// TIA Portal V20 export
DATA_BLOCK "HmiInterface"   // DB159
// stored: Access Published, MemoryReserve 100, Namespace Unit1.Em3
   VAR
      em : "LAF_typeEmInterface";
      cm : "Unit1.Em3.typeCmHmiInterface";
      topTapeLoading : "LER_typeSequenceInterface";
      topTapeAttachment : "LER_typeSequenceInterface";
      topTapeFixStage : "LER_typeSequenceInterface";
      TopTapeIdleTime : "Unit1.Em3.typeTopTapeIdleTimeHmiInterface";
      topTapeCuttingCount : "LER_typeAlarmCounterInterface";
      cmTopTapeJRDetect : "LBC_typeDigitalSignalInterface";
      cmTopTapeDiameter : "LBC_typeDigitalSignalInterface";
   END_VAR
   VAR RETAIN
      cmTopTapeAxisX { S7_SetPoint := 'True'} : "LBC_typeAxis64PosInterface";
      cmTopTapeAxisY { S7_SetPoint := 'True'} : "LBC_typeAxis64PosInterface";
   END_VAR
   VAR
      cmTopTapeLoadingBwdFwd : "LBC_typeTwoWayActuatorInterface";
      cmTopTapeLoadingClampOpenClose : "LBC_typeTwoWayActuatorInterface";
      cmTopTapeCutterUpDown : "LBC_typeTwoWayActuatorInterface";
      cmTopTapeCutterClampUpDown : "LBC_typeTwoWayActuatorInterface";
      cmTopTapeTensionBwdFwd : "LBC_typeTwoWayActuatorInterface";
      cmTopTapeAttachmentUpDown : "LBC_typeTwoWayActuatorInterface";
      cmTopTapeClampTopLeftUpDown : "LBC_typeTwoWayActuatorInterface";
      cmTopTapeClampTopCenterUpDown : "LBC_typeTwoWayActuatorInterface";
      cmTopTapeClampTopRightUpDown : "LBC_typeTwoWayActuatorInterface";
      cmTopTapeClampBtmDownUp : "LBC_typeTwoWayActuatorInterface";
      cmTopTapeClampAllOpenClose : "LBC_typeTwoWayActuatorInterface";
      cmTopTapeAttachmentVaccumOffOn : "LBC_typeTwoWayActuatorInterface";
      cmQrHandyReader : "LER_typeDM8700Interface";
      intCondition : "Unit1.Em3.typeIntConditionHmiInterface";
   END_VAR
BEGIN
   em.interlinkMode.link := FALSE;
   em.interlinkMode.unlink := FALSE;
   em.interlinkMode.isLinked := TRUE;
   em.commands.enable := FALSE;
   em.commands.acknowledge := FALSE;
   em.commands.disableAlarms := FALSE;
   em.commands.activateSimulation := FALSE;
   em.commands.home := FALSE;
   em.commands.moveToInitialPosition := FALSE;
   em.commands.directModeControl := 16#0000_0002;
   em.commands.directStateControl := 16#0000_0002;
   em.status.enabled := FALSE;
   em.status.acknowledgeActive := FALSE;
   em.status.alarmsDisabled := FALSE;
   em.status.simulationActive := FALSE;
   em.status.safetyReleased := TRUE;
   em.status.initialized := FALSE;
   em.status.homed := TRUE;
   em.status.safeState := FALSE;
   em.status.stateComplete := FALSE;
   em.alarms.error := FALSE;
   em.alarms.warning := FALSE;
   em.alarms.info := FALSE;
   TopTapeIdleTime.processCount := T#300M;
   topTapeCuttingCount.referenceDesignator := WSTRING#'Em3 Top Tape Cutting Count';
   topTapeCuttingCount.ProcessValue.faultCount := 50000;
   topTapeCuttingCount.SetValue.faultCount := 50000;
   cmTopTapeJRDetect.commands.refreshConfiguration := FALSE;
   cmTopTapeJRDetect.commands.editConfiguration := FALSE;
   cmTopTapeJRDetect.commands.saveConfiguration := FALSE;
   cmTopTapeJRDetect.commands.reset := FALSE;
   cmTopTapeJRDetect.monitoring.enable := TRUE;
   cmTopTapeJRDetect.monitoring.referenceDesignator := WSTRING#'DigitalSignal';
   cmTopTapeJRDetect.monitoring.simulation := FALSE;
   cmTopTapeJRDetect.monitoring.processValue := FALSE;
   cmTopTapeJRDetect.monitoring.error := FALSE;
   cmTopTapeJRDetect.monitoring.status := 16#0000;
   cmTopTapeJRDetect.configuration.referenceDesignator := WSTRING#'DigitalSignal';
   cmTopTapeJRDetect.configuration.onDelay := T#0MS;
   cmTopTapeJRDetect.configuration.offDelay := T#0MS;
   cmTopTapeJRDetect.configuration.default := FALSE;
   cmTopTapeJRDetect.configuration.invertProcessValue := FALSE;
   cmTopTapeJRDetect.configuration.disableAlarms := FALSE;
   cmTopTapeDiameter.commands.refreshConfiguration := FALSE;
   cmTopTapeDiameter.commands.editConfiguration := FALSE;
   cmTopTapeDiameter.commands.saveConfiguration := FALSE;
   cmTopTapeDiameter.commands.reset := FALSE;
   cmTopTapeDiameter.monitoring.enable := TRUE;
   cmTopTapeDiameter.monitoring.referenceDesignator := WSTRING#'DigitalSignal';
   cmTopTapeDiameter.monitoring.simulation := FALSE;
   cmTopTapeDiameter.monitoring.processValue := FALSE;
   cmTopTapeDiameter.monitoring.error := FALSE;
   cmTopTapeDiameter.monitoring.status := 16#0000;
   cmTopTapeDiameter.configuration.referenceDesignator := WSTRING#'DigitalSignal';
   cmTopTapeDiameter.configuration.onDelay := T#0MS;
   cmTopTapeDiameter.configuration.offDelay := T#0MS;
   cmTopTapeDiameter.configuration.default := FALSE;
   cmTopTapeDiameter.configuration.invertProcessValue := FALSE;
   cmTopTapeDiameter.configuration.disableAlarms := FALSE;
   cmTopTapeAxisX.commandConfiguration.generalSettings.stopOnError := TRUE;
   cmTopTapeAxisX.commandConfiguration.generalSettings.resetWithRestart := FALSE;
   cmTopTapeAxisX.commandConfiguration.generalSettings.abortWaitingSyncCmd := TRUE;
   cmTopTapeAxisX.commandConfiguration.power.startMode := 1;
   cmTopTapeAxisX.commandConfiguration.power.stopMode := 0;
   cmTopTapeAxisX.commandConfiguration.power.syncMotionSimulation := FALSE;
   cmTopTapeAxisX.commandConfiguration.power.syncMotionSimulationExtendedMode := -1;
   cmTopTapeAxisX.commandConfiguration.jog.velocity := 1.0;
   cmTopTapeAxisX.commandConfiguration.jog.acceleration := 100.0;
   cmTopTapeAxisX.commandConfiguration.jog.deceleration := 100.0;
   cmTopTapeAxisX.commandConfiguration.jog.jerk := 0.0;
   cmTopTapeAxisX.commandConfiguration.jog.positionControlled := TRUE;
   cmTopTapeAxisX.commandConfiguration.jog.increment := 0.0;
   cmTopTapeAxisX.commandConfiguration.jog.mode := 0;
   cmTopTapeAxisX.commandConfiguration.moveVelocity.velocity := 10.0;
   cmTopTapeAxisX.commandConfiguration.moveVelocity.acceleration := 1000.0;
   cmTopTapeAxisX.commandConfiguration.moveVelocity.deceleration := 1000.0;
   cmTopTapeAxisX.commandConfiguration.moveVelocity.jerk := -1.0;
   cmTopTapeAxisX.commandConfiguration.moveVelocity.direction := 0;
   cmTopTapeAxisX.commandConfiguration.moveVelocity.positionControlled := TRUE;
   cmTopTapeAxisX.commandConfiguration.moveVelocity.velocityChangeOnTheFly := FALSE;
   cmTopTapeAxisX.commandConfiguration.stop.deceleration := -1.0;
   cmTopTapeAxisX.commandConfiguration.stop.jerk := -1.0;
   cmTopTapeAxisX.commandConfiguration.stop.abortAcceleration := FALSE;
   cmTopTapeAxisX.commandConfiguration.fastStop.deceleration := -1.0;
   cmTopTapeAxisX.commandConfiguration.fastStop.jerk := -1.0;
   cmTopTapeAxisX.commandConfiguration.fastStop.abortAcceleration := FALSE;
   cmTopTapeAxisX.commandConfiguration.fastStop.replaceStopPossible := FALSE;
   cmTopTapeAxisX.commandConfiguration.torqueLimiting.limit := -1.0;
   cmTopTapeAxisX.commandConfiguration.torqueLimiting.mode := 0;
   cmTopTapeAxisX.commandConfiguration.homing.position := 0.0;
   cmTopTapeAxisX.commandConfiguration.homing.mode := 3;
   cmTopTapeAxisX.commandConfiguration.homing.sensor := 0;
   cmTopTapeAxisX.commandConfiguration.homing.extendedMode := -1;
   cmTopTapeAxisX.commandConfiguration.homing.extendedModeTorqueLimit := 0.0;
   cmTopTapeAxisX.commandConfiguration.homing.extendedModeTargetPosition := 0.0;
   cmTopTapeAxisX.commandConfiguration.posRelative.distance := 0.0;
   cmTopTapeAxisX.commandConfiguration.posRelative.velocity := -1.0;
   cmTopTapeAxisX.commandConfiguration.posRelative.acceleration := -1.0;
   cmTopTapeAxisX.commandConfiguration.posRelative.deceleration := -1.0;
   cmTopTapeAxisX.commandConfiguration.posRelative.jerk := -1.0;
   cmTopTapeAxisX.commandConfiguration.posRelative.direction := 0;
   cmTopTapeAxisX.commandConfiguration.posAbsolute.position := 0.0;
   cmTopTapeAxisX.commandConfiguration.posAbsolute.velocity := -1.0;
   cmTopTapeAxisX.commandConfiguration.posAbsolute.acceleration := -1.0;
   cmTopTapeAxisX.commandConfiguration.posAbsolute.deceleration := -1.0;
   cmTopTapeAxisX.commandConfiguration.posAbsolute.jerk := -1.0;
   cmTopTapeAxisX.commandConfiguration.posAbsolute.direction := 1;
   cmTopTapeAxisX.commandConfiguration.posAbsolute.positionChangeOnTheFly := FALSE;
   cmTopTapeAxisX.commandConfiguration.posAbsolute.velocityChangeOnTheFly := FALSE;
   cmTopTapeAxisX.commandConfiguration.posSuperimposed.distance := 0.0;
   cmTopTapeAxisX.commandConfiguration.posSuperimposed.velocityDiff := -1.0;
   cmTopTapeAxisX.commandConfiguration.posSuperimposed.acceleration := -1.0;
   cmTopTapeAxisX.commandConfiguration.posSuperimposed.deceleration := -1.0;
   cmTopTapeAxisX.commandConfiguration.posSuperimposed.jerk := -1.0;
   cmTopTapeAxisX.commandConfiguration.posSuperimposed.direction := 0;
   cmTopTapeAxisX.commandConfiguration.haltSuperimposed.deceleration := -1.0;
   cmTopTapeAxisX.commandConfiguration.haltSuperimposed.jerk := -1.0;
   cmTopTapeAxisX.commandConfiguration.haltSuperimposed.abortAcceleration := FALSE;
   cmTopTapeAxisX.commandConfiguration.gearInRelative.ratioNumerator := 1;
   cmTopTapeAxisX.commandConfiguration.gearInRelative.ratioDenominator := 1;
   cmTopTapeAxisX.commandConfiguration.gearInRelative.acceleration := -1.0;
   cmTopTapeAxisX.commandConfiguration.gearInRelative.deceleration := -1.0;
   cmTopTapeAxisX.commandConfiguration.gearInRelative.jerk := -1.0;
   cmTopTapeAxisX.commandConfiguration.gearInRelative.ratioChangeOnTheFly := FALSE;
   cmTopTapeAxisX.commandConfiguration.gearInAbsolute.ratioNumerator := 1;
   cmTopTapeAxisX.commandConfiguration.gearInAbsolute.ratioDenominator := 1;
   cmTopTapeAxisX.commandConfiguration.gearInAbsolute.masterSyncPosition := 0.0;
   cmTopTapeAxisX.commandConfiguration.gearInAbsolute.slaveSyncPosition := 0.0;
   cmTopTapeAxisX.commandConfiguration.gearInAbsolute.syncProfileReference := 1;
   cmTopTapeAxisX.commandConfiguration.gearInAbsolute.masterStartDistance := 0.0;
   cmTopTapeAxisX.commandConfiguration.gearInAbsolute.velocity := -1.0;
   cmTopTapeAxisX.commandConfiguration.gearInAbsolute.acceleration := -1.0;
   cmTopTapeAxisX.commandConfiguration.gearInAbsolute.deceleration := -1.0;
   cmTopTapeAxisX.commandConfiguration.gearInAbsolute.jerk := -1.0;
   cmTopTapeAxisX.commandConfiguration.gearInAbsolute.syncDirection := 1;
   cmTopTapeAxisX.commandConfiguration.gearInAbsolute.ratioChangeOnTheFly := FALSE;
   cmTopTapeAxisX.commandConfiguration.gearInVelocity.continuousUpdate := FALSE;
   cmTopTapeAxisX.commandConfiguration.gearInVelocity.ratioNumerator := 1;
   cmTopTapeAxisX.commandConfiguration.gearInVelocity.ratioDenominator := 1;
   cmTopTapeAxisX.commandConfiguration.gearInVelocity.acceleration := -1.0;
   cmTopTapeAxisX.commandConfiguration.gearInVelocity.deceleration := -1.0;
   cmTopTapeAxisX.commandConfiguration.gearInVelocity.jerk := -1.0;
   cmTopTapeAxisX.commandConfiguration.gearInVelocity.positionControlled := FALSE;
   cmTopTapeAxisX.commandConfiguration.camIn.masterOffset := 0.0;
   cmTopTapeAxisX.commandConfiguration.camIn.slaveOffset := 0.0;
   cmTopTapeAxisX.commandConfiguration.camIn.masterScaling := 1.0;
   cmTopTapeAxisX.commandConfiguration.camIn.slaveScaling := 1.0;
   cmTopTapeAxisX.commandConfiguration.camIn.masterSyncPosition := 0.0;
   cmTopTapeAxisX.commandConfiguration.camIn.syncProfileReference := 1;
   cmTopTapeAxisX.commandConfiguration.camIn.masterStartDistance := 0.0;
   cmTopTapeAxisX.commandConfiguration.camIn.velocity := -1.0;
   cmTopTapeAxisX.commandConfiguration.camIn.acceleration := -1.0;
   cmTopTapeAxisX.commandConfiguration.camIn.deceleration := -1.0;
   cmTopTapeAxisX.commandConfiguration.camIn.jerk := -1.0;
   cmTopTapeAxisX.commandConfiguration.camIn.applicationMode := 0;
   cmTopTapeAxisX.commandConfiguration.camIn.syncDirection := 1;
   cmTopTapeAxisX.commandConfiguration.gearOutCamOut.slavePosition := 0.0;
   cmTopTapeAxisX.commandConfiguration.gearOutCamOut.syncProfileReference := 1;
   cmTopTapeAxisX.commandConfiguration.gearOutCamOut.masterStopDistance := 0.0;
   cmTopTapeAxisX.commandConfiguration.gearOutCamOut.deceleration := -1.0;
   cmTopTapeAxisX.commandConfiguration.gearOutCamOut.jerk := -1.0;
   cmTopTapeAxisX.commandConfiguration.gearOutCamOut.syncOutDirection := 3;
   cmTopTapeAxisX.commandConfiguration.gearOutCamOut.gearOutCamOutMode := -1;
   cmTopTapeAxisX.commandConfiguration.phasing.phaseShift := 0.0;
   cmTopTapeAxisX.commandConfiguration.phasing.velocity := -1.0;
   cmTopTapeAxisX.commandConfiguration.phasing.acceleration := -1.0;
   cmTopTapeAxisX.commandConfiguration.phasing.deceleration := -1.0;
   cmTopTapeAxisX.commandConfiguration.phasing.jerk := -1.0;
   cmTopTapeAxisX.commandConfiguration.phasing.profileReference := 0;
   cmTopTapeAxisX.commandConfiguration.phasing.phasingDistance := 0.0;
   cmTopTapeAxisX.commandConfiguration.phasing.startPosition := 0.0;
   cmTopTapeAxisX.commandConfiguration.phasing.direction := 3;
   cmTopTapeAxisX.commandConfiguration.phasing.phaseAbsolute := TRUE;
   cmTopTapeAxisX.commandConfiguration.phasing.phaseShiftChangeOnTheFly := FALSE;
   cmTopTapeAxisX.commandConfiguration.offset.offset := 0.0;
   cmTopTapeAxisX.commandConfiguration.offset.profileReference := 1;
   cmTopTapeAxisX.commandConfiguration.offset.offsetDistance := 0.0;
   cmTopTapeAxisX.commandConfiguration.offset.startPosition := 0.0;
   cmTopTapeAxisX.commandConfiguration.offset.direction := 3;
   cmTopTapeAxisX.commandConfiguration.offset.offsetAbsolute := TRUE;
   cmTopTapeAxisX.commandConfiguration.offset.offsetChangeOnTheFly := FALSE;
   cmTopTapeAxisX.commands.enableMasterControl := FALSE;
   cmTopTapeAxisX.commands.enableAxis := FALSE;
   cmTopTapeAxisX.commands.resetAxis := FALSE;
   cmTopTapeAxisX.commands.openBrake := FALSE;
   cmTopTapeAxisX.commands.jogForward := FALSE;
   cmTopTapeAxisX.commands.jogBackward := FALSE;
   cmTopTapeAxisX.commands.moveVelocity := FALSE;
   cmTopTapeAxisX.commands.stop := FALSE;
   cmTopTapeAxisX.commands.fastStop := FALSE;
   cmTopTapeAxisX.commands.torqueLimiting := FALSE;
   cmTopTapeAxisX.commands.homing := FALSE;
   cmTopTapeAxisX.commands.posRelative := FALSE;
   cmTopTapeAxisX.commands.posAbsolute := FALSE;
   cmTopTapeAxisX.commands.posSuperimposed := FALSE;
   cmTopTapeAxisX.commands.haltSuperimposed := FALSE;
   cmTopTapeAxisX.commands.selectSetPosition := 0;
   cmTopTapeAxisX.commands.uploadParameters := FALSE;
   cmTopTapeAxisX.commands.refreshConfiguration := FALSE;
   cmTopTapeAxisX.commands.editConfiguration := FALSE;
   cmTopTapeAxisX.commands.saveConfiguration := FALSE;
   cmTopTapeAxisX.commands.uploadCurrentTorque := FALSE;
   cmTopTapeAxisX.commands.reset := FALSE;
   cmTopTapeAxisX.monitoring.enable := TRUE;
   cmTopTapeAxisX.monitoring.referenceDesignator := WSTRING#'TOP TAPING X-Axis';
   cmTopTapeAxisX.monitoring.enabled := TRUE;
   cmTopTapeAxisX.monitoring.enableManualCmds := TRUE;
   cmTopTapeAxisX.monitoring.reset := FALSE;
   cmTopTapeAxisX.monitoring.resetAxis := FALSE;
   cmTopTapeAxisX.monitoring.enableAxis := FALSE;
   cmTopTapeAxisX.monitoring.openBrake := FALSE;
   cmTopTapeAxisX.monitoring.jogBackward := FALSE;
   cmTopTapeAxisX.monitoring.jogForward := FALSE;
   cmTopTapeAxisX.monitoring.moveVelocity := FALSE;
   cmTopTapeAxisX.monitoring.stop := FALSE;
   cmTopTapeAxisX.monitoring.fastStop := FALSE;
   cmTopTapeAxisX.monitoring.torqueLimiting := FALSE;
   cmTopTapeAxisX.monitoring.homing := FALSE;
   cmTopTapeAxisX.monitoring.posRelative := FALSE;
   cmTopTapeAxisX.monitoring.posAbsolute := TRUE;
   cmTopTapeAxisX.monitoring.posSuperimposed := FALSE;
   cmTopTapeAxisX.monitoring.haltSuperimposed := FALSE;
   cmTopTapeAxisX.monitoring.brakeOpened := FALSE;
   cmTopTapeAxisX.monitoring.axisEnabled := FALSE;
   cmTopTapeAxisX.monitoring.resetActive := FALSE;
   cmTopTapeAxisX.monitoring.inVelocity := FALSE;
   cmTopTapeAxisX.monitoring.inLimitation := FALSE;
   cmTopTapeAxisX.monitoring.inClamping := FALSE;
   cmTopTapeAxisX.monitoring.startSync := FALSE;
   cmTopTapeAxisX.monitoring.inSync := FALSE;
   cmTopTapeAxisX.monitoring.inSimulation := FALSE;
   cmTopTapeAxisX.monitoring.jogSelected := FALSE;
   cmTopTapeAxisX.monitoring.moveVelocitySelected := FALSE;
   cmTopTapeAxisX.monitoring.stopSelected := FALSE;
   cmTopTapeAxisX.monitoring.fastStopSelected := FALSE;
   cmTopTapeAxisX.monitoring.torqueLimitingSelected := FALSE;
   cmTopTapeAxisX.monitoring.homingSelected := FALSE;
   cmTopTapeAxisX.monitoring.posRelativeSelected := FALSE;
   cmTopTapeAxisX.monitoring.posAbsoluteSelected := TRUE;
   cmTopTapeAxisX.monitoring.posSuperimposedSelected := FALSE;
   cmTopTapeAxisX.monitoring.haltSuperimposedSelected := FALSE;
   cmTopTapeAxisX.monitoring.commandBusy := FALSE;
   cmTopTapeAxisX.monitoring.commandDone := TRUE;
   cmTopTapeAxisX.monitoring.commandAborted := FALSE;
   cmTopTapeAxisX.monitoring.homingCommandBusy := FALSE;
   cmTopTapeAxisX.monitoring.homingCommandDone := FALSE;
   cmTopTapeAxisX.monitoring.homingCommandAborted := FALSE;
   cmTopTapeAxisX.monitoring.superimposedBusy := FALSE;
   cmTopTapeAxisX.monitoring.superimposedDone := FALSE;
   cmTopTapeAxisX.monitoring.superimposedAborted := FALSE;
   cmTopTapeAxisX.monitoring.selectSetPosition := 0;
   cmTopTapeAxisX.monitoring.selectionController := FALSE;
   cmTopTapeAxisX.monitoring.interlockGeneral := FALSE;
   cmTopTapeAxisX.monitoring.interlockJogForward := TRUE;
   cmTopTapeAxisX.monitoring.interlockJogBackward := TRUE;
   cmTopTapeAxisX.monitoring.interlockWarningGeneral := FALSE;
   cmTopTapeAxisX.monitoring.interlockWarningJogForward := FALSE;
   cmTopTapeAxisX.monitoring.interlockWarningJogBackward := FALSE;
   cmTopTapeAxisX.monitoring.valid := TRUE;
   cmTopTapeAxisX.monitoring.busy := TRUE;
   cmTopTapeAxisX.monitoring.error := FALSE;
   cmTopTapeAxisX.monitoring.status := 16#7101;
   cmTopTapeAxisX.monitoring.subfunctionStatus := 16#0000;
   cmTopTapeAxisX.monitoring.actualPosition := -0.999;
   cmTopTapeAxisX.monitoring.actualSpeed := 0.0;
   cmTopTapeAxisX.monitoring.speedUnit := 1062;
   cmTopTapeAxisX.monitoring.positionUnit := 1013;
   cmTopTapeAxisX.monitoring.axisType := 1;
   cmTopTapeAxisX.monitoring.maxVelocity := 1000.0;
   cmTopTapeAxisX.monitoring.actualCurrent := 0.0;
   cmTopTapeAxisX.monitoring.actualTorque := 0.0;
   cmTopTapeAxisX.monitoring.velocityOverrideEnabled := FALSE;
   cmTopTapeAxisX.monitoring.sinaParaError := FALSE;
   cmTopTapeAxisX.monitoring.sinaParaStatus := 16#0000_0000;
   cmTopTapeAxisX.configuration.referenceDesignator := WSTRING#'TOP TAPING X-Axis';
   cmTopTapeAxisX.configuration.disableAlarms := FALSE;
   cmTopTapeAxisX.configuration.masterControlPopUp := TRUE;
   cmTopTapeAxisX.configuration.setPositions[3..9].position := 0.0;
   cmTopTapeAxisX.configuration.setPositions[11..15].position := 0.0;
   cmTopTapeAxisX.configuration.setPositions[3..9].velocity := 0.0;
   cmTopTapeAxisX.configuration.setPositions[11..15].velocity := 0.0;
   cmTopTapeAxisX.configuration.setPositions[3..9].acceleration := 0.0;
   cmTopTapeAxisX.configuration.setPositions[11..15].acceleration := 0.0;
   cmTopTapeAxisX.configuration.setPositions[3..9].deceleration := 0.0;
   cmTopTapeAxisX.configuration.setPositions[11..15].deceleration := 0.0;
   cmTopTapeAxisX.configuration.setPositions[0]."name" := 'Wait [Tape Get]';
   cmTopTapeAxisX.configuration.setPositions[1]."name" := 'Tape1 Put';
   cmTopTapeAxisX.configuration.setPositions[2]."name" := 'Tape2 Put';
   cmTopTapeAxisX.configuration.setPositions[3]."name" := 'Remain Attachment';
   cmTopTapeAxisX.configuration.setPositions[4..8]."name" := '';
   cmTopTapeAxisX.configuration.setPositions[9]."name" := 'tapePutZone';
   cmTopTapeAxisX.configuration.setPositions[10]."name" := 'Tape Put Zone';
   cmTopTapeAxisX.configuration.setPositions[11..15]."name" := '';
   cmTopTapeAxisY.commandConfiguration.generalSettings.stopOnError := TRUE;
   cmTopTapeAxisY.commandConfiguration.generalSettings.resetWithRestart := FALSE;
   cmTopTapeAxisY.commandConfiguration.generalSettings.abortWaitingSyncCmd := TRUE;
   cmTopTapeAxisY.commandConfiguration.power.startMode := 1;
   cmTopTapeAxisY.commandConfiguration.power.stopMode := 0;
   cmTopTapeAxisY.commandConfiguration.power.syncMotionSimulation := FALSE;
   cmTopTapeAxisY.commandConfiguration.power.syncMotionSimulationExtendedMode := -1;
   cmTopTapeAxisY.commandConfiguration.jog.velocity := 20.0;
   cmTopTapeAxisY.commandConfiguration.jog.acceleration := 200.0;
   cmTopTapeAxisY.commandConfiguration.jog.deceleration := 200.0;
   cmTopTapeAxisY.commandConfiguration.jog.jerk := 0.0;
   cmTopTapeAxisY.commandConfiguration.jog.positionControlled := TRUE;
   cmTopTapeAxisY.commandConfiguration.jog.increment := 0.0;
   cmTopTapeAxisY.commandConfiguration.jog.mode := 0;
   cmTopTapeAxisY.commandConfiguration.moveVelocity.velocity := 1.0;
   cmTopTapeAxisY.commandConfiguration.moveVelocity.acceleration := -1.0;
   cmTopTapeAxisY.commandConfiguration.moveVelocity.deceleration := -1.0;
   cmTopTapeAxisY.commandConfiguration.moveVelocity.jerk := -1.0;
   cmTopTapeAxisY.commandConfiguration.moveVelocity.direction := 0;
   cmTopTapeAxisY.commandConfiguration.moveVelocity.positionControlled := TRUE;
   cmTopTapeAxisY.commandConfiguration.moveVelocity.velocityChangeOnTheFly := FALSE;
   cmTopTapeAxisY.commandConfiguration.stop.deceleration := -1.0;
   cmTopTapeAxisY.commandConfiguration.stop.jerk := -1.0;
   cmTopTapeAxisY.commandConfiguration.stop.abortAcceleration := FALSE;
   cmTopTapeAxisY.commandConfiguration.fastStop.deceleration := -1.0;
   cmTopTapeAxisY.commandConfiguration.fastStop.jerk := -1.0;
   cmTopTapeAxisY.commandConfiguration.fastStop.abortAcceleration := FALSE;
   cmTopTapeAxisY.commandConfiguration.fastStop.replaceStopPossible := FALSE;
   cmTopTapeAxisY.commandConfiguration.torqueLimiting.limit := -1.0;
   cmTopTapeAxisY.commandConfiguration.torqueLimiting.mode := 0;
   cmTopTapeAxisY.commandConfiguration.homing.position := 0.0;
   cmTopTapeAxisY.commandConfiguration.homing.mode := 3;
   cmTopTapeAxisY.commandConfiguration.homing.sensor := 0;
   cmTopTapeAxisY.commandConfiguration.homing.extendedMode := -1;
   cmTopTapeAxisY.commandConfiguration.homing.extendedModeTorqueLimit := 0.0;
   cmTopTapeAxisY.commandConfiguration.homing.extendedModeTargetPosition := 0.0;
   cmTopTapeAxisY.commandConfiguration.posRelative.distance := 0.0;
   cmTopTapeAxisY.commandConfiguration.posRelative.velocity := -1.0;
   cmTopTapeAxisY.commandConfiguration.posRelative.acceleration := -1.0;
   cmTopTapeAxisY.commandConfiguration.posRelative.deceleration := -1.0;
   cmTopTapeAxisY.commandConfiguration.posRelative.jerk := -1.0;
   cmTopTapeAxisY.commandConfiguration.posRelative.direction := 0;
   cmTopTapeAxisY.commandConfiguration.posAbsolute.position := 0.0;
   cmTopTapeAxisY.commandConfiguration.posAbsolute.velocity := -1.0;
   cmTopTapeAxisY.commandConfiguration.posAbsolute.acceleration := -1.0;
   cmTopTapeAxisY.commandConfiguration.posAbsolute.deceleration := -1.0;
   cmTopTapeAxisY.commandConfiguration.posAbsolute.jerk := -1.0;
   cmTopTapeAxisY.commandConfiguration.posAbsolute.direction := 1;
   cmTopTapeAxisY.commandConfiguration.posAbsolute.positionChangeOnTheFly := FALSE;
   cmTopTapeAxisY.commandConfiguration.posAbsolute.velocityChangeOnTheFly := FALSE;
   cmTopTapeAxisY.commandConfiguration.posSuperimposed.distance := 0.0;
   cmTopTapeAxisY.commandConfiguration.posSuperimposed.velocityDiff := -1.0;
   cmTopTapeAxisY.commandConfiguration.posSuperimposed.acceleration := -1.0;
   cmTopTapeAxisY.commandConfiguration.posSuperimposed.deceleration := -1.0;
   cmTopTapeAxisY.commandConfiguration.posSuperimposed.jerk := -1.0;
   cmTopTapeAxisY.commandConfiguration.posSuperimposed.direction := 0;
   cmTopTapeAxisY.commandConfiguration.haltSuperimposed.deceleration := -1.0;
   cmTopTapeAxisY.commandConfiguration.haltSuperimposed.jerk := -1.0;
   cmTopTapeAxisY.commandConfiguration.haltSuperimposed.abortAcceleration := FALSE;
   cmTopTapeAxisY.commandConfiguration.gearInRelative.ratioNumerator := 1;
   cmTopTapeAxisY.commandConfiguration.gearInRelative.ratioDenominator := 1;
   cmTopTapeAxisY.commandConfiguration.gearInRelative.acceleration := -1.0;
   cmTopTapeAxisY.commandConfiguration.gearInRelative.deceleration := -1.0;
   cmTopTapeAxisY.commandConfiguration.gearInRelative.jerk := -1.0;
   cmTopTapeAxisY.commandConfiguration.gearInRelative.ratioChangeOnTheFly := FALSE;
   cmTopTapeAxisY.commandConfiguration.gearInAbsolute.ratioNumerator := 1;
   cmTopTapeAxisY.commandConfiguration.gearInAbsolute.ratioDenominator := 1;
   cmTopTapeAxisY.commandConfiguration.gearInAbsolute.masterSyncPosition := 0.0;
   cmTopTapeAxisY.commandConfiguration.gearInAbsolute.slaveSyncPosition := 0.0;
   cmTopTapeAxisY.commandConfiguration.gearInAbsolute.syncProfileReference := 1;
   cmTopTapeAxisY.commandConfiguration.gearInAbsolute.masterStartDistance := 0.0;
   cmTopTapeAxisY.commandConfiguration.gearInAbsolute.velocity := -1.0;
   cmTopTapeAxisY.commandConfiguration.gearInAbsolute.acceleration := -1.0;
   cmTopTapeAxisY.commandConfiguration.gearInAbsolute.deceleration := -1.0;
   cmTopTapeAxisY.commandConfiguration.gearInAbsolute.jerk := -1.0;
   cmTopTapeAxisY.commandConfiguration.gearInAbsolute.syncDirection := 1;
   cmTopTapeAxisY.commandConfiguration.gearInAbsolute.ratioChangeOnTheFly := FALSE;
   cmTopTapeAxisY.commandConfiguration.gearInVelocity.continuousUpdate := FALSE;
   cmTopTapeAxisY.commandConfiguration.gearInVelocity.ratioNumerator := 1;
   cmTopTapeAxisY.commandConfiguration.gearInVelocity.ratioDenominator := 1;
   cmTopTapeAxisY.commandConfiguration.gearInVelocity.acceleration := -1.0;
   cmTopTapeAxisY.commandConfiguration.gearInVelocity.deceleration := -1.0;
   cmTopTapeAxisY.commandConfiguration.gearInVelocity.jerk := -1.0;
   cmTopTapeAxisY.commandConfiguration.gearInVelocity.positionControlled := FALSE;
   cmTopTapeAxisY.commandConfiguration.camIn.masterOffset := 0.0;
   cmTopTapeAxisY.commandConfiguration.camIn.slaveOffset := 0.0;
   cmTopTapeAxisY.commandConfiguration.camIn.masterScaling := 1.0;
   cmTopTapeAxisY.commandConfiguration.camIn.slaveScaling := 1.0;
   cmTopTapeAxisY.commandConfiguration.camIn.masterSyncPosition := 0.0;
   cmTopTapeAxisY.commandConfiguration.camIn.syncProfileReference := 1;
   cmTopTapeAxisY.commandConfiguration.camIn.masterStartDistance := 0.0;
   cmTopTapeAxisY.commandConfiguration.camIn.velocity := -1.0;
   cmTopTapeAxisY.commandConfiguration.camIn.acceleration := -1.0;
   cmTopTapeAxisY.commandConfiguration.camIn.deceleration := -1.0;
   cmTopTapeAxisY.commandConfiguration.camIn.jerk := -1.0;
   cmTopTapeAxisY.commandConfiguration.camIn.applicationMode := 0;
   cmTopTapeAxisY.commandConfiguration.camIn.syncDirection := 1;
   cmTopTapeAxisY.commandConfiguration.gearOutCamOut.slavePosition := 0.0;
   cmTopTapeAxisY.commandConfiguration.gearOutCamOut.syncProfileReference := 1;
   cmTopTapeAxisY.commandConfiguration.gearOutCamOut.masterStopDistance := 0.0;
   cmTopTapeAxisY.commandConfiguration.gearOutCamOut.deceleration := -1.0;
   cmTopTapeAxisY.commandConfiguration.gearOutCamOut.jerk := -1.0;
   cmTopTapeAxisY.commandConfiguration.gearOutCamOut.syncOutDirection := 3;
   cmTopTapeAxisY.commandConfiguration.gearOutCamOut.gearOutCamOutMode := -1;
   cmTopTapeAxisY.commandConfiguration.phasing.phaseShift := 0.0;
   cmTopTapeAxisY.commandConfiguration.phasing.velocity := -1.0;
   cmTopTapeAxisY.commandConfiguration.phasing.acceleration := -1.0;
   cmTopTapeAxisY.commandConfiguration.phasing.deceleration := -1.0;
   cmTopTapeAxisY.commandConfiguration.phasing.jerk := -1.0;
   cmTopTapeAxisY.commandConfiguration.phasing.profileReference := 0;
   cmTopTapeAxisY.commandConfiguration.phasing.phasingDistance := 0.0;
   cmTopTapeAxisY.commandConfiguration.phasing.startPosition := 0.0;
   cmTopTapeAxisY.commandConfiguration.phasing.direction := 3;
   cmTopTapeAxisY.commandConfiguration.phasing.phaseAbsolute := TRUE;
   cmTopTapeAxisY.commandConfiguration.phasing.phaseShiftChangeOnTheFly := FALSE;
   cmTopTapeAxisY.commandConfiguration.offset.offset := 0.0;
   cmTopTapeAxisY.commandConfiguration.offset.profileReference := 1;
   cmTopTapeAxisY.commandConfiguration.offset.offsetDistance := 0.0;
   cmTopTapeAxisY.commandConfiguration.offset.startPosition := 0.0;
   cmTopTapeAxisY.commandConfiguration.offset.direction := 3;
   cmTopTapeAxisY.commandConfiguration.offset.offsetAbsolute := TRUE;
   cmTopTapeAxisY.commandConfiguration.offset.offsetChangeOnTheFly := FALSE;
   cmTopTapeAxisY.commands.enableMasterControl := FALSE;
   cmTopTapeAxisY.commands.enableAxis := FALSE;
   cmTopTapeAxisY.commands.resetAxis := FALSE;
   cmTopTapeAxisY.commands.openBrake := FALSE;
   cmTopTapeAxisY.commands.jogForward := FALSE;
   cmTopTapeAxisY.commands.jogBackward := FALSE;
   cmTopTapeAxisY.commands.moveVelocity := FALSE;
   cmTopTapeAxisY.commands.stop := FALSE;
   cmTopTapeAxisY.commands.fastStop := FALSE;
   cmTopTapeAxisY.commands.torqueLimiting := FALSE;
   cmTopTapeAxisY.commands.homing := FALSE;
   cmTopTapeAxisY.commands.posRelative := FALSE;
   cmTopTapeAxisY.commands.posAbsolute := FALSE;
   cmTopTapeAxisY.commands.posSuperimposed := FALSE;
   cmTopTapeAxisY.commands.haltSuperimposed := FALSE;
   cmTopTapeAxisY.commands.selectSetPosition := 0;
   cmTopTapeAxisY.commands.uploadParameters := FALSE;
   cmTopTapeAxisY.commands.refreshConfiguration := FALSE;
   cmTopTapeAxisY.commands.editConfiguration := FALSE;
   cmTopTapeAxisY.commands.saveConfiguration := FALSE;
   cmTopTapeAxisY.commands.uploadCurrentTorque := FALSE;
   cmTopTapeAxisY.commands.reset := FALSE;
   cmTopTapeAxisY.monitoring.enable := TRUE;
   cmTopTapeAxisY.monitoring.referenceDesignator := WSTRING#'TOP TAPING Y-Axis';
   cmTopTapeAxisY.monitoring.enabled := TRUE;
   cmTopTapeAxisY.monitoring.enableManualCmds := TRUE;
   cmTopTapeAxisY.monitoring.reset := FALSE;
   cmTopTapeAxisY.monitoring.resetAxis := FALSE;
   cmTopTapeAxisY.monitoring.enableAxis := FALSE;
   cmTopTapeAxisY.monitoring.openBrake := FALSE;
   cmTopTapeAxisY.monitoring.jogBackward := FALSE;
   cmTopTapeAxisY.monitoring.jogForward := FALSE;
   cmTopTapeAxisY.monitoring.moveVelocity := FALSE;
   cmTopTapeAxisY.monitoring.stop := FALSE;
   cmTopTapeAxisY.monitoring.fastStop := FALSE;
   cmTopTapeAxisY.monitoring.torqueLimiting := FALSE;
   cmTopTapeAxisY.monitoring.homing := FALSE;
   cmTopTapeAxisY.monitoring.posRelative := FALSE;
   cmTopTapeAxisY.monitoring.posAbsolute := TRUE;
   cmTopTapeAxisY.monitoring.posSuperimposed := FALSE;
   cmTopTapeAxisY.monitoring.haltSuperimposed := FALSE;
   cmTopTapeAxisY.monitoring.brakeOpened := FALSE;
   cmTopTapeAxisY.monitoring.axisEnabled := FALSE;
   cmTopTapeAxisY.monitoring.resetActive := FALSE;
   cmTopTapeAxisY.monitoring.inVelocity := FALSE;
   cmTopTapeAxisY.monitoring.inLimitation := FALSE;
   cmTopTapeAxisY.monitoring.inClamping := FALSE;
   cmTopTapeAxisY.monitoring.startSync := FALSE;
   cmTopTapeAxisY.monitoring.inSync := FALSE;
   cmTopTapeAxisY.monitoring.inSimulation := FALSE;
   cmTopTapeAxisY.monitoring.jogSelected := FALSE;
   cmTopTapeAxisY.monitoring.moveVelocitySelected := FALSE;
   cmTopTapeAxisY.monitoring.stopSelected := FALSE;
   cmTopTapeAxisY.monitoring.fastStopSelected := FALSE;
   cmTopTapeAxisY.monitoring.torqueLimitingSelected := FALSE;
   cmTopTapeAxisY.monitoring.homingSelected := FALSE;
   cmTopTapeAxisY.monitoring.posRelativeSelected := FALSE;
   cmTopTapeAxisY.monitoring.posAbsoluteSelected := TRUE;
   cmTopTapeAxisY.monitoring.posSuperimposedSelected := FALSE;
   cmTopTapeAxisY.monitoring.haltSuperimposedSelected := FALSE;
   cmTopTapeAxisY.monitoring.commandBusy := FALSE;
   cmTopTapeAxisY.monitoring.commandDone := TRUE;
   cmTopTapeAxisY.monitoring.commandAborted := FALSE;
   cmTopTapeAxisY.monitoring.homingCommandBusy := FALSE;
   cmTopTapeAxisY.monitoring.homingCommandDone := FALSE;
   cmTopTapeAxisY.monitoring.homingCommandAborted := FALSE;
   cmTopTapeAxisY.monitoring.superimposedBusy := FALSE;
   cmTopTapeAxisY.monitoring.superimposedDone := FALSE;
   cmTopTapeAxisY.monitoring.superimposedAborted := FALSE;
   cmTopTapeAxisY.monitoring.selectSetPosition := 0;
   cmTopTapeAxisY.monitoring.selectionController := FALSE;
   cmTopTapeAxisY.monitoring.interlockGeneral := FALSE;
   cmTopTapeAxisY.monitoring.interlockJogForward := TRUE;
   cmTopTapeAxisY.monitoring.interlockJogBackward := TRUE;
   cmTopTapeAxisY.monitoring.interlockWarningGeneral := FALSE;
   cmTopTapeAxisY.monitoring.interlockWarningJogForward := FALSE;
   cmTopTapeAxisY.monitoring.interlockWarningJogBackward := FALSE;
   cmTopTapeAxisY.monitoring.valid := TRUE;
   cmTopTapeAxisY.monitoring.busy := TRUE;
   cmTopTapeAxisY.monitoring.error := FALSE;
   cmTopTapeAxisY.monitoring.status := 16#7101;
   cmTopTapeAxisY.monitoring.subfunctionStatus := 16#0000;
   cmTopTapeAxisY.monitoring.actualPosition := 293.001;
   cmTopTapeAxisY.monitoring.actualSpeed := 0.0;
   cmTopTapeAxisY.monitoring.speedUnit := 1062;
   cmTopTapeAxisY.monitoring.positionUnit := 1013;
   cmTopTapeAxisY.monitoring.axisType := 1;
   cmTopTapeAxisY.monitoring.maxVelocity := 1000.0;
   cmTopTapeAxisY.monitoring.actualCurrent := 0.0;
   cmTopTapeAxisY.monitoring.actualTorque := 0.0;
   cmTopTapeAxisY.monitoring.velocityOverrideEnabled := FALSE;
   cmTopTapeAxisY.monitoring.sinaParaError := FALSE;
   cmTopTapeAxisY.monitoring.sinaParaStatus := 16#0000_0000;
   cmTopTapeAxisY.configuration.referenceDesignator := WSTRING#'TOP TAPING Y-Axis';
   cmTopTapeAxisY.configuration.disableAlarms := FALSE;
   cmTopTapeAxisY.configuration.masterControlPopUp := TRUE;
   cmTopTapeAxisY.configuration.setPositions[3..7].position := 0.0;
   cmTopTapeAxisY.configuration.setPositions[11..15].position := 0.0;
   cmTopTapeAxisY.configuration.setPositions[3..7].velocity := 0.0;
   cmTopTapeAxisY.configuration.setPositions[11..15].velocity := 0.0;
   cmTopTapeAxisY.configuration.setPositions[3..7].acceleration := 0.0;
   cmTopTapeAxisY.configuration.setPositions[11..15].acceleration := 0.0;
   cmTopTapeAxisY.configuration.setPositions[3..7].deceleration := 0.0;
   cmTopTapeAxisY.configuration.setPositions[11..15].deceleration := 0.0;
   cmTopTapeAxisY.configuration.setPositions[0]."name" := 'Wait [Taping]';
   cmTopTapeAxisY.configuration.setPositions[1]."name" := 'Load';
   cmTopTapeAxisY.configuration.setPositions[2]."name" := 'Unload';
   cmTopTapeAxisY.configuration.setPositions[3..8]."name" := '';
   cmTopTapeAxisY.configuration.setPositions[9]."name" := 'Load Zone';
   cmTopTapeAxisY.configuration.setPositions[10]."name" := 'Unload Zone';
   cmTopTapeAxisY.configuration.setPositions[11..15]."name" := '';
   cmTopTapeLoadingBwdFwd.commands.refreshConfiguration := FALSE;
   cmTopTapeLoadingBwdFwd.commands.editConfiguration := FALSE;
   cmTopTapeLoadingBwdFwd.commands.saveConfiguration := FALSE;
   cmTopTapeLoadingBwdFwd.commands.reset := FALSE;
   cmTopTapeLoadingBwdFwd.commands.commandHomePos := FALSE;
   cmTopTapeLoadingBwdFwd.commands.commandWorkPos := FALSE;
   cmTopTapeLoadingBwdFwd.monitoring.enable := TRUE;
   cmTopTapeLoadingBwdFwd.monitoring.referenceDesignator := WSTRING#'T.TAPE LOADING';
   cmTopTapeLoadingBwdFwd.monitoring.commandHomePos := FALSE;
   cmTopTapeLoadingBwdFwd.monitoring.commandWorkPos := FALSE;
   cmTopTapeLoadingBwdFwd.monitoring.goToHomePos := TRUE;
   cmTopTapeLoadingBwdFwd.monitoring.goToWorkPos := FALSE;
   cmTopTapeLoadingBwdFwd.monitoring.inHomePos := TRUE;
   cmTopTapeLoadingBwdFwd.monitoring.inWorkPos := FALSE;
   cmTopTapeLoadingBwdFwd.monitoring.reset := FALSE;
   cmTopTapeLoadingBwdFwd.monitoring.enableManualCmds := TRUE;
   cmTopTapeLoadingBwdFwd.monitoring.error := FALSE;
   cmTopTapeLoadingBwdFwd.monitoring.interlockHomePos := TRUE;
   cmTopTapeLoadingBwdFwd.monitoring.interlockWorkPos := TRUE;
   cmTopTapeLoadingBwdFwd.monitoring.status := 16#7004;
   cmTopTapeLoadingBwdFwd.monitoring.interlockWarningWorkPos := FALSE;
   cmTopTapeLoadingBwdFwd.monitoring.interlockWarningHomePos := FALSE;
   cmTopTapeLoadingBwdFwd.configuration.referenceDesignator := WSTRING#'T.TAPE LOADING';
   cmTopTapeLoadingBwdFwd.configuration.monitoringLeavingFeedback := T#5S;
   cmTopTapeLoadingBwdFwd.configuration.monitoringReachingFeedback := T#5S;
   cmTopTapeLoadingBwdFwd.configuration.monitoringDiscrepancy := T#5S;
   cmTopTapeLoadingBwdFwd.configuration.setOutputHomeContinuously := TRUE;
   cmTopTapeLoadingBwdFwd.configuration.setOutputWorkContinuously := TRUE;
   cmTopTapeLoadingBwdFwd.configuration.disableHomeCommand := FALSE;
   cmTopTapeLoadingBwdFwd.configuration.disableFeedbackHomePos := FALSE;
   cmTopTapeLoadingBwdFwd.configuration.disableFeedbackWorkPos := FALSE;
   cmTopTapeLoadingBwdFwd.configuration.disableAlarms := FALSE;
   cmTopTapeLoadingBwdFwd.configuration.resetOutputsOnError := FALSE;
   cmTopTapeLoadingBwdFwd.configuration.allwaysWaitOnReachingTime := FALSE;
   cmTopTapeLoadingClampOpenClose.commands.refreshConfiguration := FALSE;
   cmTopTapeLoadingClampOpenClose.commands.editConfiguration := FALSE;
   cmTopTapeLoadingClampOpenClose.commands.saveConfiguration := FALSE;
   cmTopTapeLoadingClampOpenClose.commands.reset := FALSE;
   cmTopTapeLoadingClampOpenClose.commands.commandHomePos := FALSE;
   cmTopTapeLoadingClampOpenClose.commands.commandWorkPos := FALSE;
   cmTopTapeLoadingClampOpenClose.monitoring.enable := TRUE;
   cmTopTapeLoadingClampOpenClose.monitoring.referenceDesignator := WSTRING#'T.TAPE LOADING CLAMP';
   cmTopTapeLoadingClampOpenClose.monitoring.commandHomePos := FALSE;
   cmTopTapeLoadingClampOpenClose.monitoring.commandWorkPos := FALSE;
   cmTopTapeLoadingClampOpenClose.monitoring.goToHomePos := FALSE;
   cmTopTapeLoadingClampOpenClose.monitoring.goToWorkPos := TRUE;
   cmTopTapeLoadingClampOpenClose.monitoring.inHomePos := FALSE;
   cmTopTapeLoadingClampOpenClose.monitoring.inWorkPos := TRUE;
   cmTopTapeLoadingClampOpenClose.monitoring.reset := FALSE;
   cmTopTapeLoadingClampOpenClose.monitoring.enableManualCmds := TRUE;
   cmTopTapeLoadingClampOpenClose.monitoring.error := FALSE;
   cmTopTapeLoadingClampOpenClose.monitoring.interlockHomePos := TRUE;
   cmTopTapeLoadingClampOpenClose.monitoring.interlockWorkPos := TRUE;
   cmTopTapeLoadingClampOpenClose.monitoring.status := 16#7006;
   cmTopTapeLoadingClampOpenClose.monitoring.interlockWarningWorkPos := FALSE;
   cmTopTapeLoadingClampOpenClose.monitoring.interlockWarningHomePos := FALSE;
   cmTopTapeLoadingClampOpenClose.configuration.referenceDesignator := WSTRING#'T.TAPE LOADING CLAMP';
   cmTopTapeLoadingClampOpenClose.configuration.monitoringLeavingFeedback := T#5S;
   cmTopTapeLoadingClampOpenClose.configuration.monitoringReachingFeedback := T#5S;
   cmTopTapeLoadingClampOpenClose.configuration.monitoringDiscrepancy := T#5S;
   cmTopTapeLoadingClampOpenClose.configuration.setOutputHomeContinuously := TRUE;
   cmTopTapeLoadingClampOpenClose.configuration.setOutputWorkContinuously := TRUE;
   cmTopTapeLoadingClampOpenClose.configuration.disableHomeCommand := FALSE;
   cmTopTapeLoadingClampOpenClose.configuration.disableFeedbackHomePos := FALSE;
   cmTopTapeLoadingClampOpenClose.configuration.disableFeedbackWorkPos := FALSE;
   cmTopTapeLoadingClampOpenClose.configuration.disableAlarms := FALSE;
   cmTopTapeLoadingClampOpenClose.configuration.resetOutputsOnError := FALSE;
   cmTopTapeLoadingClampOpenClose.configuration.allwaysWaitOnReachingTime := FALSE;
   cmTopTapeCutterUpDown.commands.refreshConfiguration := FALSE;
   cmTopTapeCutterUpDown.commands.editConfiguration := FALSE;
   cmTopTapeCutterUpDown.commands.saveConfiguration := FALSE;
   cmTopTapeCutterUpDown.commands.reset := FALSE;
   cmTopTapeCutterUpDown.commands.commandHomePos := FALSE;
   cmTopTapeCutterUpDown.commands.commandWorkPos := FALSE;
   cmTopTapeCutterUpDown.monitoring.enable := TRUE;
   cmTopTapeCutterUpDown.monitoring.referenceDesignator := WSTRING#'T.TAPE CUTTER';
   cmTopTapeCutterUpDown.monitoring.commandHomePos := FALSE;
   cmTopTapeCutterUpDown.monitoring.commandWorkPos := FALSE;
   cmTopTapeCutterUpDown.monitoring.goToHomePos := TRUE;
   cmTopTapeCutterUpDown.monitoring.goToWorkPos := FALSE;
   cmTopTapeCutterUpDown.monitoring.inHomePos := TRUE;
   cmTopTapeCutterUpDown.monitoring.inWorkPos := FALSE;
   cmTopTapeCutterUpDown.monitoring.reset := FALSE;
   cmTopTapeCutterUpDown.monitoring.enableManualCmds := TRUE;
   cmTopTapeCutterUpDown.monitoring.error := FALSE;
   cmTopTapeCutterUpDown.monitoring.interlockHomePos := TRUE;
   cmTopTapeCutterUpDown.monitoring.interlockWorkPos := TRUE;
   cmTopTapeCutterUpDown.monitoring.status := 16#7004;
   cmTopTapeCutterUpDown.monitoring.interlockWarningWorkPos := FALSE;
   cmTopTapeCutterUpDown.monitoring.interlockWarningHomePos := FALSE;
   cmTopTapeCutterUpDown.configuration.referenceDesignator := WSTRING#'T.TAPE CUTTER';
   cmTopTapeCutterUpDown.configuration.monitoringLeavingFeedback := T#5S;
   cmTopTapeCutterUpDown.configuration.monitoringReachingFeedback := T#5S;
   cmTopTapeCutterUpDown.configuration.monitoringDiscrepancy := T#5S;
   cmTopTapeCutterUpDown.configuration.setOutputHomeContinuously := TRUE;
   cmTopTapeCutterUpDown.configuration.setOutputWorkContinuously := TRUE;
   cmTopTapeCutterUpDown.configuration.disableHomeCommand := FALSE;
   cmTopTapeCutterUpDown.configuration.disableFeedbackHomePos := FALSE;
   cmTopTapeCutterUpDown.configuration.disableFeedbackWorkPos := FALSE;
   cmTopTapeCutterUpDown.configuration.disableAlarms := FALSE;
   cmTopTapeCutterUpDown.configuration.resetOutputsOnError := FALSE;
   cmTopTapeCutterUpDown.configuration.allwaysWaitOnReachingTime := FALSE;
   cmTopTapeCutterClampUpDown.commands.refreshConfiguration := FALSE;
   cmTopTapeCutterClampUpDown.commands.editConfiguration := FALSE;
   cmTopTapeCutterClampUpDown.commands.saveConfiguration := FALSE;
   cmTopTapeCutterClampUpDown.commands.reset := FALSE;
   cmTopTapeCutterClampUpDown.commands.commandHomePos := FALSE;
   cmTopTapeCutterClampUpDown.commands.commandWorkPos := FALSE;
   cmTopTapeCutterClampUpDown.monitoring.enable := TRUE;
   cmTopTapeCutterClampUpDown.monitoring.referenceDesignator := WSTRING#'T.TAPE CUTTER CLAMP';
   cmTopTapeCutterClampUpDown.monitoring.commandHomePos := FALSE;
   cmTopTapeCutterClampUpDown.monitoring.commandWorkPos := FALSE;
   cmTopTapeCutterClampUpDown.monitoring.goToHomePos := FALSE;
   cmTopTapeCutterClampUpDown.monitoring.goToWorkPos := TRUE;
   cmTopTapeCutterClampUpDown.monitoring.inHomePos := FALSE;
   cmTopTapeCutterClampUpDown.monitoring.inWorkPos := TRUE;
   cmTopTapeCutterClampUpDown.monitoring.reset := FALSE;
   cmTopTapeCutterClampUpDown.monitoring.enableManualCmds := TRUE;
   cmTopTapeCutterClampUpDown.monitoring.error := FALSE;
   cmTopTapeCutterClampUpDown.monitoring.interlockHomePos := TRUE;
   cmTopTapeCutterClampUpDown.monitoring.interlockWorkPos := TRUE;
   cmTopTapeCutterClampUpDown.monitoring.status := 16#7006;
   cmTopTapeCutterClampUpDown.monitoring.interlockWarningWorkPos := FALSE;
   cmTopTapeCutterClampUpDown.monitoring.interlockWarningHomePos := FALSE;
   cmTopTapeCutterClampUpDown.configuration.referenceDesignator := WSTRING#'T.TAPE CUTTER CLAMP';
   cmTopTapeCutterClampUpDown.configuration.monitoringLeavingFeedback := T#5S;
   cmTopTapeCutterClampUpDown.configuration.monitoringReachingFeedback := T#5S;
   cmTopTapeCutterClampUpDown.configuration.monitoringDiscrepancy := T#5S;
   cmTopTapeCutterClampUpDown.configuration.setOutputHomeContinuously := TRUE;
   cmTopTapeCutterClampUpDown.configuration.setOutputWorkContinuously := TRUE;
   cmTopTapeCutterClampUpDown.configuration.disableHomeCommand := FALSE;
   cmTopTapeCutterClampUpDown.configuration.disableFeedbackHomePos := FALSE;
   cmTopTapeCutterClampUpDown.configuration.disableFeedbackWorkPos := FALSE;
   cmTopTapeCutterClampUpDown.configuration.disableAlarms := FALSE;
   cmTopTapeCutterClampUpDown.configuration.resetOutputsOnError := FALSE;
   cmTopTapeCutterClampUpDown.configuration.allwaysWaitOnReachingTime := FALSE;
   cmTopTapeTensionBwdFwd.commands.refreshConfiguration := FALSE;
   cmTopTapeTensionBwdFwd.commands.editConfiguration := FALSE;
   cmTopTapeTensionBwdFwd.commands.saveConfiguration := FALSE;
   cmTopTapeTensionBwdFwd.commands.reset := FALSE;
   cmTopTapeTensionBwdFwd.commands.commandHomePos := FALSE;
   cmTopTapeTensionBwdFwd.commands.commandWorkPos := FALSE;
   cmTopTapeTensionBwdFwd.monitoring.enable := TRUE;
   cmTopTapeTensionBwdFwd.monitoring.referenceDesignator := WSTRING#'T.TAPE TENSION';
   cmTopTapeTensionBwdFwd.monitoring.commandHomePos := FALSE;
   cmTopTapeTensionBwdFwd.monitoring.commandWorkPos := FALSE;
   cmTopTapeTensionBwdFwd.monitoring.goToHomePos := TRUE;
   cmTopTapeTensionBwdFwd.monitoring.goToWorkPos := FALSE;
   cmTopTapeTensionBwdFwd.monitoring.inHomePos := TRUE;
   cmTopTapeTensionBwdFwd.monitoring.inWorkPos := FALSE;
   cmTopTapeTensionBwdFwd.monitoring.reset := FALSE;
   cmTopTapeTensionBwdFwd.monitoring.enableManualCmds := TRUE;
   cmTopTapeTensionBwdFwd.monitoring.error := FALSE;
   cmTopTapeTensionBwdFwd.monitoring.interlockHomePos := TRUE;
   cmTopTapeTensionBwdFwd.monitoring.interlockWorkPos := TRUE;
   cmTopTapeTensionBwdFwd.monitoring.status := 16#7004;
   cmTopTapeTensionBwdFwd.monitoring.interlockWarningWorkPos := FALSE;
   cmTopTapeTensionBwdFwd.monitoring.interlockWarningHomePos := FALSE;
   cmTopTapeTensionBwdFwd.configuration.referenceDesignator := WSTRING#'T.TAPE TENSION';
   cmTopTapeTensionBwdFwd.configuration.monitoringLeavingFeedback := T#5S;
   cmTopTapeTensionBwdFwd.configuration.monitoringReachingFeedback := T#5S;
   cmTopTapeTensionBwdFwd.configuration.monitoringDiscrepancy := T#5S;
   cmTopTapeTensionBwdFwd.configuration.setOutputHomeContinuously := TRUE;
   cmTopTapeTensionBwdFwd.configuration.setOutputWorkContinuously := TRUE;
   cmTopTapeTensionBwdFwd.configuration.disableHomeCommand := FALSE;
   cmTopTapeTensionBwdFwd.configuration.disableFeedbackHomePos := FALSE;
   cmTopTapeTensionBwdFwd.configuration.disableFeedbackWorkPos := FALSE;
   cmTopTapeTensionBwdFwd.configuration.disableAlarms := FALSE;
   cmTopTapeTensionBwdFwd.configuration.resetOutputsOnError := FALSE;
   cmTopTapeTensionBwdFwd.configuration.allwaysWaitOnReachingTime := FALSE;
   cmTopTapeAttachmentUpDown.commands.refreshConfiguration := FALSE;
   cmTopTapeAttachmentUpDown.commands.editConfiguration := FALSE;
   cmTopTapeAttachmentUpDown.commands.saveConfiguration := FALSE;
   cmTopTapeAttachmentUpDown.commands.reset := FALSE;
   cmTopTapeAttachmentUpDown.commands.commandHomePos := FALSE;
   cmTopTapeAttachmentUpDown.commands.commandWorkPos := FALSE;
   cmTopTapeAttachmentUpDown.monitoring.enable := TRUE;
   cmTopTapeAttachmentUpDown.monitoring.referenceDesignator := WSTRING#'T.TAPE ATTACHMENT';
   cmTopTapeAttachmentUpDown.monitoring.commandHomePos := FALSE;
   cmTopTapeAttachmentUpDown.monitoring.commandWorkPos := FALSE;
   cmTopTapeAttachmentUpDown.monitoring.goToHomePos := TRUE;
   cmTopTapeAttachmentUpDown.monitoring.goToWorkPos := FALSE;
   cmTopTapeAttachmentUpDown.monitoring.inHomePos := TRUE;
   cmTopTapeAttachmentUpDown.monitoring.inWorkPos := FALSE;
   cmTopTapeAttachmentUpDown.monitoring.reset := FALSE;
   cmTopTapeAttachmentUpDown.monitoring.enableManualCmds := TRUE;
   cmTopTapeAttachmentUpDown.monitoring.error := FALSE;
   cmTopTapeAttachmentUpDown.monitoring.interlockHomePos := TRUE;
   cmTopTapeAttachmentUpDown.monitoring.interlockWorkPos := TRUE;
   cmTopTapeAttachmentUpDown.monitoring.status := 16#7004;
   cmTopTapeAttachmentUpDown.monitoring.interlockWarningWorkPos := FALSE;
   cmTopTapeAttachmentUpDown.monitoring.interlockWarningHomePos := FALSE;
   cmTopTapeAttachmentUpDown.configuration.referenceDesignator := WSTRING#'T.TAPE ATTACHMENT';
   cmTopTapeAttachmentUpDown.configuration.monitoringLeavingFeedback := T#5S;
   cmTopTapeAttachmentUpDown.configuration.monitoringReachingFeedback := T#5S;
   cmTopTapeAttachmentUpDown.configuration.monitoringDiscrepancy := T#5S;
   cmTopTapeAttachmentUpDown.configuration.setOutputHomeContinuously := TRUE;
   cmTopTapeAttachmentUpDown.configuration.setOutputWorkContinuously := TRUE;
   cmTopTapeAttachmentUpDown.configuration.disableHomeCommand := FALSE;
   cmTopTapeAttachmentUpDown.configuration.disableFeedbackHomePos := FALSE;
   cmTopTapeAttachmentUpDown.configuration.disableFeedbackWorkPos := FALSE;
   cmTopTapeAttachmentUpDown.configuration.disableAlarms := FALSE;
   cmTopTapeAttachmentUpDown.configuration.resetOutputsOnError := FALSE;
   cmTopTapeAttachmentUpDown.configuration.allwaysWaitOnReachingTime := FALSE;
   cmTopTapeClampTopLeftUpDown.commands.refreshConfiguration := FALSE;
   cmTopTapeClampTopLeftUpDown.commands.editConfiguration := FALSE;
   cmTopTapeClampTopLeftUpDown.commands.saveConfiguration := FALSE;
   cmTopTapeClampTopLeftUpDown.commands.reset := FALSE;
   cmTopTapeClampTopLeftUpDown.commands.commandHomePos := FALSE;
   cmTopTapeClampTopLeftUpDown.commands.commandWorkPos := FALSE;
   cmTopTapeClampTopLeftUpDown.monitoring.enable := TRUE;
   cmTopTapeClampTopLeftUpDown.monitoring.referenceDesignator := WSTRING#'T.TAPE CLAMP TOP LEFT';
   cmTopTapeClampTopLeftUpDown.monitoring.commandHomePos := FALSE;
   cmTopTapeClampTopLeftUpDown.monitoring.commandWorkPos := FALSE;
   cmTopTapeClampTopLeftUpDown.monitoring.goToHomePos := TRUE;
   cmTopTapeClampTopLeftUpDown.monitoring.goToWorkPos := FALSE;
   cmTopTapeClampTopLeftUpDown.monitoring.inHomePos := TRUE;
   cmTopTapeClampTopLeftUpDown.monitoring.inWorkPos := FALSE;
   cmTopTapeClampTopLeftUpDown.monitoring.reset := FALSE;
   cmTopTapeClampTopLeftUpDown.monitoring.enableManualCmds := TRUE;
   cmTopTapeClampTopLeftUpDown.monitoring.error := FALSE;
   cmTopTapeClampTopLeftUpDown.monitoring.interlockHomePos := TRUE;
   cmTopTapeClampTopLeftUpDown.monitoring.interlockWorkPos := TRUE;
   cmTopTapeClampTopLeftUpDown.monitoring.status := 16#7004;
   cmTopTapeClampTopLeftUpDown.monitoring.interlockWarningWorkPos := FALSE;
   cmTopTapeClampTopLeftUpDown.monitoring.interlockWarningHomePos := FALSE;
   cmTopTapeClampTopLeftUpDown.configuration.referenceDesignator := WSTRING#'T.TAPE CLAMP TOP LEFT';
   cmTopTapeClampTopLeftUpDown.configuration.monitoringLeavingFeedback := T#5S;
   cmTopTapeClampTopLeftUpDown.configuration.monitoringReachingFeedback := T#5S;
   cmTopTapeClampTopLeftUpDown.configuration.monitoringDiscrepancy := T#5S;
   cmTopTapeClampTopLeftUpDown.configuration.setOutputHomeContinuously := TRUE;
   cmTopTapeClampTopLeftUpDown.configuration.setOutputWorkContinuously := TRUE;
   cmTopTapeClampTopLeftUpDown.configuration.disableHomeCommand := FALSE;
   cmTopTapeClampTopLeftUpDown.configuration.disableFeedbackHomePos := FALSE;
   cmTopTapeClampTopLeftUpDown.configuration.disableFeedbackWorkPos := FALSE;
   cmTopTapeClampTopLeftUpDown.configuration.disableAlarms := FALSE;
   cmTopTapeClampTopLeftUpDown.configuration.resetOutputsOnError := FALSE;
   cmTopTapeClampTopLeftUpDown.configuration.allwaysWaitOnReachingTime := FALSE;
   cmTopTapeClampTopCenterUpDown.commands.refreshConfiguration := FALSE;
   cmTopTapeClampTopCenterUpDown.commands.editConfiguration := FALSE;
   cmTopTapeClampTopCenterUpDown.commands.saveConfiguration := FALSE;
   cmTopTapeClampTopCenterUpDown.commands.reset := FALSE;
   cmTopTapeClampTopCenterUpDown.commands.commandHomePos := FALSE;
   cmTopTapeClampTopCenterUpDown.commands.commandWorkPos := FALSE;
   cmTopTapeClampTopCenterUpDown.monitoring.enable := TRUE;
   cmTopTapeClampTopCenterUpDown.monitoring.referenceDesignator := WSTRING#'T.TAPE CLAMP TOP CENTER';
   cmTopTapeClampTopCenterUpDown.monitoring.commandHomePos := FALSE;
   cmTopTapeClampTopCenterUpDown.monitoring.commandWorkPos := FALSE;
   cmTopTapeClampTopCenterUpDown.monitoring.goToHomePos := TRUE;
   cmTopTapeClampTopCenterUpDown.monitoring.goToWorkPos := FALSE;
   cmTopTapeClampTopCenterUpDown.monitoring.inHomePos := TRUE;
   cmTopTapeClampTopCenterUpDown.monitoring.inWorkPos := FALSE;
   cmTopTapeClampTopCenterUpDown.monitoring.reset := FALSE;
   cmTopTapeClampTopCenterUpDown.monitoring.enableManualCmds := TRUE;
   cmTopTapeClampTopCenterUpDown.monitoring.error := FALSE;
   cmTopTapeClampTopCenterUpDown.monitoring.interlockHomePos := TRUE;
   cmTopTapeClampTopCenterUpDown.monitoring.interlockWorkPos := TRUE;
   cmTopTapeClampTopCenterUpDown.monitoring.status := 16#7004;
   cmTopTapeClampTopCenterUpDown.monitoring.interlockWarningWorkPos := FALSE;
   cmTopTapeClampTopCenterUpDown.monitoring.interlockWarningHomePos := FALSE;
   cmTopTapeClampTopCenterUpDown.configuration.referenceDesignator := WSTRING#'T.TAPE CLAMP TOP CENTER';
   cmTopTapeClampTopCenterUpDown.configuration.monitoringLeavingFeedback := T#5S;
   cmTopTapeClampTopCenterUpDown.configuration.monitoringReachingFeedback := T#5S;
   cmTopTapeClampTopCenterUpDown.configuration.monitoringDiscrepancy := T#5S;
   cmTopTapeClampTopCenterUpDown.configuration.setOutputHomeContinuously := TRUE;
   cmTopTapeClampTopCenterUpDown.configuration.setOutputWorkContinuously := TRUE;
   cmTopTapeClampTopCenterUpDown.configuration.disableHomeCommand := FALSE;
   cmTopTapeClampTopCenterUpDown.configuration.disableFeedbackHomePos := FALSE;
   cmTopTapeClampTopCenterUpDown.configuration.disableFeedbackWorkPos := FALSE;
   cmTopTapeClampTopCenterUpDown.configuration.disableAlarms := FALSE;
   cmTopTapeClampTopCenterUpDown.configuration.resetOutputsOnError := FALSE;
   cmTopTapeClampTopCenterUpDown.configuration.allwaysWaitOnReachingTime := FALSE;
   cmTopTapeClampTopRightUpDown.commands.refreshConfiguration := FALSE;
   cmTopTapeClampTopRightUpDown.commands.editConfiguration := FALSE;
   cmTopTapeClampTopRightUpDown.commands.saveConfiguration := FALSE;
   cmTopTapeClampTopRightUpDown.commands.reset := FALSE;
   cmTopTapeClampTopRightUpDown.commands.commandHomePos := FALSE;
   cmTopTapeClampTopRightUpDown.commands.commandWorkPos := FALSE;
   cmTopTapeClampTopRightUpDown.monitoring.enable := TRUE;
   cmTopTapeClampTopRightUpDown.monitoring.referenceDesignator := WSTRING#'T.TAPE CLAMP TOP';
   cmTopTapeClampTopRightUpDown.monitoring.commandHomePos := FALSE;
   cmTopTapeClampTopRightUpDown.monitoring.commandWorkPos := FALSE;
   cmTopTapeClampTopRightUpDown.monitoring.goToHomePos := TRUE;
   cmTopTapeClampTopRightUpDown.monitoring.goToWorkPos := FALSE;
   cmTopTapeClampTopRightUpDown.monitoring.inHomePos := TRUE;
   cmTopTapeClampTopRightUpDown.monitoring.inWorkPos := FALSE;
   cmTopTapeClampTopRightUpDown.monitoring.reset := FALSE;
   cmTopTapeClampTopRightUpDown.monitoring.enableManualCmds := TRUE;
   cmTopTapeClampTopRightUpDown.monitoring.error := FALSE;
   cmTopTapeClampTopRightUpDown.monitoring.interlockHomePos := TRUE;
   cmTopTapeClampTopRightUpDown.monitoring.interlockWorkPos := TRUE;
   cmTopTapeClampTopRightUpDown.monitoring.status := 16#7004;
   cmTopTapeClampTopRightUpDown.monitoring.interlockWarningWorkPos := FALSE;
   cmTopTapeClampTopRightUpDown.monitoring.interlockWarningHomePos := FALSE;
   cmTopTapeClampTopRightUpDown.configuration.referenceDesignator := WSTRING#'T.TAPE CLAMP TOP';
   cmTopTapeClampTopRightUpDown.configuration.monitoringLeavingFeedback := T#5S;
   cmTopTapeClampTopRightUpDown.configuration.monitoringReachingFeedback := T#5S;
   cmTopTapeClampTopRightUpDown.configuration.monitoringDiscrepancy := T#5S;
   cmTopTapeClampTopRightUpDown.configuration.setOutputHomeContinuously := TRUE;
   cmTopTapeClampTopRightUpDown.configuration.setOutputWorkContinuously := TRUE;
   cmTopTapeClampTopRightUpDown.configuration.disableHomeCommand := FALSE;
   cmTopTapeClampTopRightUpDown.configuration.disableFeedbackHomePos := FALSE;
   cmTopTapeClampTopRightUpDown.configuration.disableFeedbackWorkPos := FALSE;
   cmTopTapeClampTopRightUpDown.configuration.disableAlarms := FALSE;
   cmTopTapeClampTopRightUpDown.configuration.resetOutputsOnError := FALSE;
   cmTopTapeClampTopRightUpDown.configuration.allwaysWaitOnReachingTime := FALSE;
   cmTopTapeClampBtmDownUp.commands.refreshConfiguration := FALSE;
   cmTopTapeClampBtmDownUp.commands.editConfiguration := FALSE;
   cmTopTapeClampBtmDownUp.commands.saveConfiguration := FALSE;
   cmTopTapeClampBtmDownUp.commands.reset := FALSE;
   cmTopTapeClampBtmDownUp.commands.commandHomePos := FALSE;
   cmTopTapeClampBtmDownUp.commands.commandWorkPos := FALSE;
   cmTopTapeClampBtmDownUp.monitoring.enable := TRUE;
   cmTopTapeClampBtmDownUp.monitoring.referenceDesignator := WSTRING#'T.TAPE CLAMP BTM';
   cmTopTapeClampBtmDownUp.monitoring.commandHomePos := FALSE;
   cmTopTapeClampBtmDownUp.monitoring.commandWorkPos := FALSE;
   cmTopTapeClampBtmDownUp.monitoring.goToHomePos := TRUE;
   cmTopTapeClampBtmDownUp.monitoring.goToWorkPos := FALSE;
   cmTopTapeClampBtmDownUp.monitoring.inHomePos := TRUE;
   cmTopTapeClampBtmDownUp.monitoring.inWorkPos := FALSE;
   cmTopTapeClampBtmDownUp.monitoring.reset := FALSE;
   cmTopTapeClampBtmDownUp.monitoring.enableManualCmds := TRUE;
   cmTopTapeClampBtmDownUp.monitoring.error := FALSE;
   cmTopTapeClampBtmDownUp.monitoring.interlockHomePos := TRUE;
   cmTopTapeClampBtmDownUp.monitoring.interlockWorkPos := TRUE;
   cmTopTapeClampBtmDownUp.monitoring.status := 16#7004;
   cmTopTapeClampBtmDownUp.monitoring.interlockWarningWorkPos := FALSE;
   cmTopTapeClampBtmDownUp.monitoring.interlockWarningHomePos := FALSE;
   cmTopTapeClampBtmDownUp.configuration.referenceDesignator := WSTRING#'T.TAPE CLAMP BTM';
   cmTopTapeClampBtmDownUp.configuration.monitoringLeavingFeedback := T#5S;
   cmTopTapeClampBtmDownUp.configuration.monitoringReachingFeedback := T#5S;
   cmTopTapeClampBtmDownUp.configuration.monitoringDiscrepancy := T#5S;
   cmTopTapeClampBtmDownUp.configuration.setOutputHomeContinuously := TRUE;
   cmTopTapeClampBtmDownUp.configuration.setOutputWorkContinuously := TRUE;
   cmTopTapeClampBtmDownUp.configuration.disableHomeCommand := FALSE;
   cmTopTapeClampBtmDownUp.configuration.disableFeedbackHomePos := FALSE;
   cmTopTapeClampBtmDownUp.configuration.disableFeedbackWorkPos := FALSE;
   cmTopTapeClampBtmDownUp.configuration.disableAlarms := FALSE;
   cmTopTapeClampBtmDownUp.configuration.resetOutputsOnError := FALSE;
   cmTopTapeClampBtmDownUp.configuration.allwaysWaitOnReachingTime := FALSE;
   cmTopTapeClampAllOpenClose.commands.refreshConfiguration := FALSE;
   cmTopTapeClampAllOpenClose.commands.editConfiguration := FALSE;
   cmTopTapeClampAllOpenClose.commands.saveConfiguration := FALSE;
   cmTopTapeClampAllOpenClose.commands.reset := FALSE;
   cmTopTapeClampAllOpenClose.commands.commandHomePos := FALSE;
   cmTopTapeClampAllOpenClose.commands.commandWorkPos := FALSE;
   cmTopTapeClampAllOpenClose.monitoring.enable := TRUE;
   cmTopTapeClampAllOpenClose.monitoring.referenceDesignator := WSTRING#'TOP CLAMP ALL';
   cmTopTapeClampAllOpenClose.monitoring.commandHomePos := FALSE;
   cmTopTapeClampAllOpenClose.monitoring.commandWorkPos := FALSE;
   cmTopTapeClampAllOpenClose.monitoring.goToHomePos := FALSE;
   cmTopTapeClampAllOpenClose.monitoring.goToWorkPos := FALSE;
   cmTopTapeClampAllOpenClose.monitoring.inHomePos := FALSE;
   cmTopTapeClampAllOpenClose.monitoring.inWorkPos := FALSE;
   cmTopTapeClampAllOpenClose.monitoring.reset := FALSE;
   cmTopTapeClampAllOpenClose.monitoring.enableManualCmds := TRUE;
   cmTopTapeClampAllOpenClose.monitoring.error := FALSE;
   cmTopTapeClampAllOpenClose.monitoring.interlockHomePos := TRUE;
   cmTopTapeClampAllOpenClose.monitoring.interlockWorkPos := TRUE;
   cmTopTapeClampAllOpenClose.monitoring.status := 16#7003;
   cmTopTapeClampAllOpenClose.monitoring.interlockWarningWorkPos := FALSE;
   cmTopTapeClampAllOpenClose.monitoring.interlockWarningHomePos := FALSE;
   cmTopTapeClampAllOpenClose.configuration.referenceDesignator := WSTRING#'TOP CLAMP ALL';
   cmTopTapeClampAllOpenClose.configuration.monitoringLeavingFeedback := T#5S;
   cmTopTapeClampAllOpenClose.configuration.monitoringReachingFeedback := T#5S;
   cmTopTapeClampAllOpenClose.configuration.monitoringDiscrepancy := T#5S;
   cmTopTapeClampAllOpenClose.configuration.setOutputHomeContinuously := TRUE;
   cmTopTapeClampAllOpenClose.configuration.setOutputWorkContinuously := TRUE;
   cmTopTapeClampAllOpenClose.configuration.disableHomeCommand := FALSE;
   cmTopTapeClampAllOpenClose.configuration.disableFeedbackHomePos := FALSE;
   cmTopTapeClampAllOpenClose.configuration.disableFeedbackWorkPos := FALSE;
   cmTopTapeClampAllOpenClose.configuration.disableAlarms := FALSE;
   cmTopTapeClampAllOpenClose.configuration.resetOutputsOnError := FALSE;
   cmTopTapeClampAllOpenClose.configuration.allwaysWaitOnReachingTime := FALSE;
   cmTopTapeAttachmentVaccumOffOn.commands.refreshConfiguration := FALSE;
   cmTopTapeAttachmentVaccumOffOn.commands.editConfiguration := FALSE;
   cmTopTapeAttachmentVaccumOffOn.commands.saveConfiguration := FALSE;
   cmTopTapeAttachmentVaccumOffOn.commands.reset := FALSE;
   cmTopTapeAttachmentVaccumOffOn.commands.commandHomePos := FALSE;
   cmTopTapeAttachmentVaccumOffOn.commands.commandWorkPos := FALSE;
   cmTopTapeAttachmentVaccumOffOn.monitoring.enable := TRUE;
   cmTopTapeAttachmentVaccumOffOn.monitoring.referenceDesignator := WSTRING#'ATTACHMENT VACUUM PRESS';
   cmTopTapeAttachmentVaccumOffOn.monitoring.commandHomePos := FALSE;
   cmTopTapeAttachmentVaccumOffOn.monitoring.commandWorkPos := FALSE;
   cmTopTapeAttachmentVaccumOffOn.monitoring.goToHomePos := FALSE;
   cmTopTapeAttachmentVaccumOffOn.monitoring.goToWorkPos := TRUE;
   cmTopTapeAttachmentVaccumOffOn.monitoring.inHomePos := FALSE;
   cmTopTapeAttachmentVaccumOffOn.monitoring.inWorkPos := TRUE;
   cmTopTapeAttachmentVaccumOffOn.monitoring.reset := FALSE;
   cmTopTapeAttachmentVaccumOffOn.monitoring.enableManualCmds := TRUE;
   cmTopTapeAttachmentVaccumOffOn.monitoring.error := FALSE;
   cmTopTapeAttachmentVaccumOffOn.monitoring.interlockHomePos := TRUE;
   cmTopTapeAttachmentVaccumOffOn.monitoring.interlockWorkPos := TRUE;
   cmTopTapeAttachmentVaccumOffOn.monitoring.status := 16#7006;
   cmTopTapeAttachmentVaccumOffOn.monitoring.interlockWarningWorkPos := FALSE;
   cmTopTapeAttachmentVaccumOffOn.monitoring.interlockWarningHomePos := FALSE;
   cmTopTapeAttachmentVaccumOffOn.configuration.referenceDesignator := WSTRING#'ATTACHMENT VACUUM PRESS';
   cmTopTapeAttachmentVaccumOffOn.configuration.monitoringLeavingFeedback := T#5S;
   cmTopTapeAttachmentVaccumOffOn.configuration.monitoringReachingFeedback := T#5S;
   cmTopTapeAttachmentVaccumOffOn.configuration.monitoringDiscrepancy := T#5S;
   cmTopTapeAttachmentVaccumOffOn.configuration.setOutputHomeContinuously := TRUE;
   cmTopTapeAttachmentVaccumOffOn.configuration.setOutputWorkContinuously := TRUE;
   cmTopTapeAttachmentVaccumOffOn.configuration.disableHomeCommand := FALSE;
   cmTopTapeAttachmentVaccumOffOn.configuration.disableFeedbackHomePos := FALSE;
   cmTopTapeAttachmentVaccumOffOn.configuration.disableFeedbackWorkPos := FALSE;
   cmTopTapeAttachmentVaccumOffOn.configuration.disableAlarms := FALSE;
   cmTopTapeAttachmentVaccumOffOn.configuration.resetOutputsOnError := FALSE;
   cmTopTapeAttachmentVaccumOffOn.configuration.allwaysWaitOnReachingTime := FALSE;
   cmQrHandyReader.commands.Trigger_SW := FALSE;
   cmQrHandyReader.commands.ID_Reset := FALSE;
   cmQrHandyReader.monitoring.Input_Status.Acquisition_Status."Trigger Ready" := FALSE;
   cmQrHandyReader.monitoring.Input_Status.Acquisition_Status."Trigger Ack" := FALSE;
   cmQrHandyReader.monitoring.Input_Status.Acquisition_Status.Acquiring := FALSE;
   cmQrHandyReader.monitoring.Input_Status.Acquisition_Status."Missed Ack" := FALSE;
   cmQrHandyReader.monitoring.Input_Status.Acquisition_Status.Reserved := FALSE;
   cmQrHandyReader.monitoring.Input_Status.Acquisition_Status.Reserved_1 := FALSE;
   cmQrHandyReader.monitoring.Input_Status.Acquisition_Status.Reserved_2 := FALSE;
   cmQrHandyReader.monitoring.Input_Status.Acquisition_Status.Reserved_3 := FALSE;
   cmQrHandyReader.monitoring.Input_Status.Acquisition_Status."Trigger ID"[0..1] := ' ';
   cmQrHandyReader.monitoring.Input_Status.Results_Status.Decoding := FALSE;
   cmQrHandyReader.monitoring.Input_Status.Results_Status."Decode Complete" := FALSE;
   cmQrHandyReader.monitoring.Input_Status.Results_Status."Result Buffer Overrun" := FALSE;
   cmQrHandyReader.monitoring.Input_Status.Results_Status."Results Available" := FALSE;
   cmQrHandyReader.monitoring.Input_Status.Results_Status.Reserved := FALSE;
   cmQrHandyReader.monitoring.Input_Status.Results_Status.Reserved_1 := FALSE;
   cmQrHandyReader.monitoring.Input_Status.Results_Status.Reserved_2 := FALSE;
   cmQrHandyReader.monitoring.Input_Status.Results_Status."General Fault" := FALSE;
   cmQrHandyReader.monitoring.Input_Status.Soft_Event_Status."Train Code Ack" := FALSE;
   cmQrHandyReader.monitoring.Input_Status.Soft_Event_Status."Train Match String Ack" := FALSE;
   cmQrHandyReader.monitoring.Input_Status.Soft_Event_Status."Train Focus Ack" := FALSE;
   cmQrHandyReader.monitoring.Input_Status.Soft_Event_Status."Train Brightness Ack" := FALSE;
   cmQrHandyReader.monitoring.Input_Status.Soft_Event_Status."Untrain Ack" := FALSE;
   cmQrHandyReader.monitoring.Input_Status.Soft_Event_Status.Reserved_1 := FALSE;
   cmQrHandyReader.monitoring.Input_Status.Soft_Event_Status."Execute DMCC Ack" := FALSE;
   cmQrHandyReader.monitoring.Input_Status.Soft_Event_Status."Set Match String Ack" := FALSE;
   cmQrHandyReader.monitoring.Input_Status.Result_Data.Result_ID[0..1] := ' ';
   cmQrHandyReader.monitoring.Input_Status.Result_Data.Result_Code[0..15] := FALSE;
   cmQrHandyReader.monitoring.Input_Status.Result_Data.Result_Extended[0..1] := ' ';
   cmQrHandyReader.monitoring.Input_Status.Result_Data.Result_Data_Length[0..1] := ' ';
   cmQrHandyReader.monitoring.Input_Status.Result_Data.Result_Data[0..253] := ' ';
   cmQrHandyReader.monitoring.Ouput_Status.Acquisition_Control."Trigger Enable" := FALSE;
   cmQrHandyReader.monitoring.Ouput_Status.Acquisition_Control.Trigger := FALSE;
   cmQrHandyReader.monitoring.Ouput_Status.Acquisition_Control.Reserved := FALSE;
   cmQrHandyReader.monitoring.Ouput_Status.Acquisition_Control.Reserved_1 := FALSE;
   cmQrHandyReader.monitoring.Ouput_Status.Acquisition_Control.Reserved_2 := FALSE;
   cmQrHandyReader.monitoring.Ouput_Status.Acquisition_Control.Reserved_3 := FALSE;
   cmQrHandyReader.monitoring.Ouput_Status.Acquisition_Control.Reserved_4 := FALSE;
   cmQrHandyReader.monitoring.Ouput_Status.Acquisition_Control.Reserved_5 := FALSE;
   cmQrHandyReader.monitoring.Ouput_Status.Results_Control."Results Buffer Enable" := FALSE;
   cmQrHandyReader.monitoring.Ouput_Status.Results_Control."Results Ack" := FALSE;
   cmQrHandyReader.monitoring.Ouput_Status.Results_Control.Reserved := FALSE;
   cmQrHandyReader.monitoring.Ouput_Status.Results_Control.Reserved_1 := FALSE;
   cmQrHandyReader.monitoring.Ouput_Status.Results_Control.Reserved_2 := FALSE;
   cmQrHandyReader.monitoring.Ouput_Status.Results_Control.Reserved_3 := FALSE;
   cmQrHandyReader.monitoring.Ouput_Status.Results_Control.Reserved_4 := FALSE;
   cmQrHandyReader.monitoring.Ouput_Status.Results_Control.Reserved_5 := FALSE;
   cmQrHandyReader.monitoring.Ouput_Status.Soft_Event_Control."Train Code" := FALSE;
   cmQrHandyReader.monitoring.Ouput_Status.Soft_Event_Control."Train MatchString" := FALSE;
   cmQrHandyReader.monitoring.Ouput_Status.Soft_Event_Control."Train Focus" := FALSE;
   cmQrHandyReader.monitoring.Ouput_Status.Soft_Event_Control.TrainBrightness := FALSE;
   cmQrHandyReader.monitoring.Ouput_Status.Soft_Event_Control.Untrain := FALSE;
   cmQrHandyReader.monitoring.Ouput_Status.Soft_Event_Control.Reserved := FALSE;
   cmQrHandyReader.monitoring.Ouput_Status.Soft_Event_Control.ExecuteDMCC := FALSE;
   cmQrHandyReader.monitoring.Ouput_Status.Soft_Event_Control."Set MatchString" := FALSE;
   cmQrHandyReader.monitoring.Ouput_Status.User_Data."User Data Option"[0..1] := ' ';
   cmQrHandyReader.monitoring.Ouput_Status.User_Data."User Data Length"[0..1] := ' ';
   cmQrHandyReader.monitoring.Ouput_Status.User_Data."User Data"[0..253] := ' ';
   cmQrHandyReader.monitoring.Result_Data_ID := '';
   cmQrHandyReader.monitoring.ReadOk := FALSE;
   cmQrHandyReader.monitoring.ReadNg := FALSE;
   cmQrHandyReader.monitoring.ReadComplete := FALSE;
   cmQrHandyReader.monitoring.Error := FALSE;
   cmQrHandyReader.configuration.Acquisition_Status_HW_ID := 0;
   cmQrHandyReader.configuration.Results_Status_HW_ID := 0;
   cmQrHandyReader.configuration.Soft_Event_Status_HW_ID := 0;
   cmQrHandyReader.configuration.Result_Data_HW_ID := 0;
   cmQrHandyReader.configuration.Acquisition_Control_HW_ID := 0;
   cmQrHandyReader.configuration.Results_Control_HW_ID := 0;
   cmQrHandyReader.configuration.Soft_Event_Control_HW_ID := 0;
   cmQrHandyReader.configuration.User_Data_HW_ID := 0;
   cmQrHandyReader.configuration.Retry_SV := 1;
   cmQrHandyReader.configuration.BCR_Type := FALSE;
END_DATA_BLOCK
